FUNCTION_BLOCK PUBLIC FB_AmericanPizzaCalifornia EXTENDS FB_AmericanPizzaMargherita
VAR_INPUT
END_VAR
VAR_OUTPUT
END_VAR
VAR
	bPepperoni	: BOOL := TRUE;
END_VAR

PROPERTY PUBLIC bHasPepperoni : BOOL
GET
bHasPepperoni := this^.bPepperoni;
END_GET
SET
this^.bPepperoni := bHasPepperoni;
END_SET
END_PROPERTY

METHOD PUBLIC GetPrice : LREAL
VAR_INPUT
END_VAR
GetPrice := SUPER^.GetPrice();
IF (THIS^.bPepperoni) THEN
	GetPrice := GetPrice + 0.4;
END_IF
END_METHOD

END_FUNCTION_BLOCK

(* stored: Version 1.1.0.1, ProductVersion 3.1.4022.12
   POU FB_AmericanPizzaCalifornia: Id {1708d268-70e2-4bce-b487-de09dbe3ebe6}, SpecialFunc None
   Property bHasPepperoni: Id {7f1e896f-d0c8-4a2b-bdb0-a5f8a47cdb09}
   Get Get: Id {4ddd5c93-f39d-446e-ba79-2e459c5831c7}
   Set Set: Id {11872f25-a0b6-4eb7-8ab6-267f6a7234d4}
   Method GetPrice: Id {b4c04cb9-2ab2-4401-a9bb-30468ed49619} *)
